FUNCTION "LGF_IntToString" : String
TITLE = LGF_IntToString
{ S7_Optimized_Access := 'TRUE' }
AUTHOR : Siemens_Digital_Industry
FAMILY : LGF
NAME : LGF_IntToString
//This function converts a variable of the data type `DInt` into a variable of the data type `String`.
   VAR_INPUT
      value : DInt;   // Double-Integer value to convert
   END_VAR

   VAR_TEMP
      tempString : String;   // Temp string for conversion from double integer
   END_VAR

   VAR CONSTANT
      CONVERT_SIZE : USInt := 0;   // Number of character positions
      CONVERT_PRECISION : USInt := 0;   // Number of decimal places
      CONVERT_FORMAT_TO_STRING : Word := 16#0000;   // Output format of the characters
      CONVERT_START_POSITION : UInt := 1;   // Character starting at which the result is written.
   END_VAR


BEGIN
	REGION BLOCK INFO HEADER
	  //===============================================================================
	  // SIEMENS AG / (c)Copyright 2017
	  //-------------------------------------------------------------------------------
	  // Title:            LGF_IntToString
	  // Comment/Function: This function converts a variable of the system data type `DInt` into a variable of the data type `String`.
	  // Library/Family:   LGF(Library General Functions)
	  // Author:           Siemens Digital Industry Support
	  // Tested with:      CPU1212C DC/DC/DC FW:V4.2
	  // Engineering:      TIA Portal V14 SP1 Upd 5
	  // Restrictions:     ENO disabled - no error handling
	  // Requirements:     PLC (S7-1200 / S7-1500)
	  //-------------------------------------------------------------------------------
	  // Change log table:
	  // Version  | Date       | Expert in charge       | Changes applied
	  //----------|------------|------------------------|------------------------------
	  // 01.00.00 | 04.07.2018 | Siemens Industry Online Support
	  //                         First released version
	  // 01.00.01 | 17.08.2018 | Siemens Industry Online Support
	  //                         Upgrade: TIA V15 Update 2
	  // 01.00.02 | 23.11.2018 | Siemens Industry Online Support
	  //                         Upgrade: TIA V15.1
	  // 01.00.05 | 07.06.2019 | Simatic Systems Support
	  //                         Standard header and block parameters update
	  //                         Program changed to VAL_STRG wrapper
	  // 01.00.06 | 30.07.2019 | Simatic Systems Support
	  //                         Add ENO handling
	  // 03.00.00 | 23.04.2020 | Simatic Systems Support | Set version to V3.0.0
	  //                         Harmonize the version of the whole library
	  // 03.00.01 | 23.02.2021 | Simatic Systems Support
	  //                         Insert documentation
	  //===============================================================================
	END_REGION Block info header

	REGION CONVERSION
	  VAL_STRG(IN     := #value,
	           SIZE   := #CONVERT_SIZE,
	           PREC   := #CONVERT_PRECISION,
	           FORMAT := #CONVERT_FORMAT_TO_STRING,
	           P      := #CONVERT_START_POSITION,
	           OUT    => #tempString);
	END_REGION

	REGION OUTPUT
	  #LGF_IntToString := #tempString;
	  // no error handling needed
	  ENO := TRUE;
	END_REGION
END_FUNCTION

